// TIA Portal V18 export
FUNCTION_BLOCK "_hmi_spot_manager"   // FB47, FBD
{ S7_Optimized_Access := 'TRUE' }
VERSION : 0.1
// stored: AutoNumber true, IsIECCheckEnabled false, IsRetainMemResEnabled false, MemoryReserve 100, SetENOAutomatically false, UDAEnableTagReadback false
   VAR_INPUT
      cur_pos_set : "typePositions";
   END_VAR
   VAR_OUTPUT
      hmi_pos_set : "typePositions";
      hmi_to_spot_allowed : Bool;
      Spot_positions_now : "typePositions";
   END_VAR
   VAR_IN_OUT
      spot_set_encoder : Bool;
      spot_set_hmi : Bool;
   END_VAR
   VAR
      spot_ws : WString;
      part_was : Int;
      spotSaver { S7_SetPoint := 'True'} : "_hmi_singleSpotManager";
   END_VAR
BEGIN

REGION Network 1
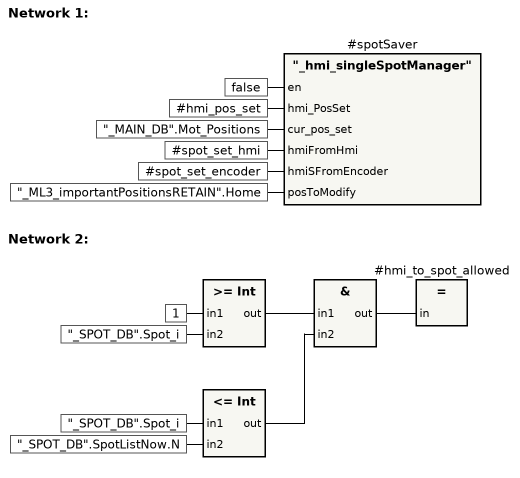
   IF false THEN
       #spotSaver(hmi_PosSet := #hmi_pos_set,   // "_hmi_singleSpotManager"
                  cur_pos_set := "_MAIN_DB".Mot_Positions,
                  hmiFromHmi := #spot_set_hmi,
                  hmiSFromEncoder := #spot_set_encoder,
                  posToModify := "_ML3_importantPositionsRETAIN".Home);
   END_IF;
END_REGION

REGION Network 2
   #hmi_to_spot_allowed := (1 >= "_SPOT_DB".Spot_i) AND ("_SPOT_DB".Spot_i <= "_SPOT_DB".SpotListNow.N);
END_REGION

REGION Network 3 (SCL)
   IF #part_was <> "_SPOT_DB".Part_selected THEN
       IF "_SPOT_DB".Part_selected > 0 AND "_SPOT_DB".Part_selected <= "_SPOT_DB".Spot_N_max THEN
           "_SPOT_DB".SpotListNow := "_SPOT_DB".Parts["_SPOT_DB".Part_selected];
       END_IF;
   ELSE
       IF "_SPOT_DB".Part_selected > 0 AND "_SPOT_DB".Part_selected < "_SPOT_DB".Spot_N_max THEN
           "_SPOT_DB".Parts["_SPOT_DB".Part_selected] := "_SPOT_DB".SpotListNow;
       END_IF;
   END_IF;

   //#Spot_positions_now :=  "_SPOT_DB".SpotListNow.pos_AR["_SPOT_DB".Spot_i];


   #part_was := "_SPOT_DB".Part_selected;
END_REGION
END_FUNCTION_BLOCK
